// TIA Portal V21 export
DATA_BLOCK "DB615"   // DB615
TITLE = DB615
{ S7_Optimized_Access := 'FALSE' }
// CIP GENERAL DB
// stored: AutoNumber false
   VAR RETAIN
      Fault : Bool;
      Running : Bool;
      Selected : Bool;
      NoCycleSelectedInterlock : Bool;
      SelectStep : Bool;
      DelayToTriggerStep : Bool;
      ResetLogic : Bool;
      ProcessOver : Bool;
      TempStep : Int;
      CurrentStep : Int;
      CycleStatus : String[60];
      StepStatus : String[60];
      StepStatusInt : Int;
      Re : Array[0..50] of Bool;
      CycleStarted { S7_SetPoint := 'True'} : "CipCycleStarted";
      CycleOver { S7_SetPoint := 'True'} : "CipCycleOver";
      CycleRunningMV : Bool;
      ApActPressure : Real;
      CheckWeightWfi : Real;
      ScanTimeForFillingWfiTemp : Int;
   END_VAR
BEGIN
END_DATA_BLOCK
